(* IEC 61131-3 sources: bcs-engineering-dsl/language/test/generating/if_test/expected, 3 files *)

(* ---- IfLogicFB_decl.st ---- *)
FUNCTION_BLOCK IfLogicFB
VAR_INPUT
    iValue1: INT;
    iValue2: INT;
    iCondition: BOOL;
END_VAR
VAR_OUTPUT
    oResult: INT;
    oStatus: STRING;
END_VAR
VAR
    tempValue: INT;
END_VAR

(* ---- IfLogicFB_impl.st ---- *)
IF iCondition THEN
    tempValue := iValue1 + iValue2;
ELSE
    tempValue := iValue1 - iValue2;
END_IF;
IF tempValue > 100 THEN
    IF iValue1 > 50 THEN
        oResult := 100;
    ELSE
        tempValue := -100;
    END_IF;
    oStatus := 'Value clamped to maximum';
ELSIF tempValue < 0 THEN
    oResult := 0;
    oStatus := 'Value clamped to minimum';
ELSE
    oResult := tempValue;
    oStatus := 'Value in range';
END_IF;

(* ---- MAIN_decl.st ---- *)
PROGRAM MAIN
VAR
    TestIfLogic_value1: INT := 75;
    TestIfLogic_value2: INT := 50;
    TestIfLogic_condition: BOOL := TRUE;
    TestIfLogic_result: INT;
    TestIfLogic_status: STRING;
    IfLogicFBInstance1: IfLogicFB;
END_VAR
